# EPICS substitutions: ek9000App/Db/EL2022.substitutions
file EL2022.template
{       pattern
        {
                TERMINAL,

        }
        {
        }
}
